// TwinCAT 3 PLC project Untitled1
// ProgramVersion: 3.1.4026.19
// libraries:
//   Tc2_Standard, * (Beckhoff Automation GmbH)
//   Tc2_System, * (Beckhoff Automation GmbH)
// project tree:
//   DUTs/ ST_Chiller_Reads.TcDUT, ST_Alarms.TcDUT (not stored), ST_Control.TcDUT, ST_Chiller_Writes.TcDUT, ST_States.TcDUT (not stored), ST_Value0.TcDUT, ST_Value1.TcDUT (not stored)
//   GVLs/ GVL_Lauda.TcGVL
//   / PlcTask.TcTTO
//   POUs/ FB_Chiller.TcPOU, MAIN.TcPOU (not stored)
// real-time tasks:
//   TASK PlcTask: cycle T#10ms, priority 20, ADS port 350
//   TASK Task_Profinet: cycle T#1ms, priority 1, ADS port 301
// I/O:
//   DEVICE Device 1 (Profinet Controller CCAT (RT)), AmsNetId 5.155.185.217.2.1
//     abx-prt [HMS Industrial Networks This Device Access Point supports RT communication Anybus X-gateway]
//       modules: Term 1 (DAP Module), Term 2 (Output 002 bytes), Term 3 (Output 032 bytes), Term 4 (Input 004 bytes), Term 5 (Input 064 bytes), Term 6 (Input 032 bytes), Term 7 (Input 016 bytes)
// variable links:
//   Untitled1/Untitled1 Instance <-> Device 1 (Profinet Controller CCAT (RT))/abx-prt
//     PlcTask Inputs/GVL_Lauda.LaudaChillerReads.ChilleStatesIn.V50011On <-> API/Term 4 (Input 004 bytes)/Subterm 6 (Input 004 bytes)/Inputs/Input[0] @bit 2
//     PlcTask Inputs/GVL_Lauda.LaudaChillerReads.ChilleStatesIn.commonFault <-> API/Term 4 (Input 004 bytes)/Subterm 6 (Input 004 bytes)/Inputs/Input[1] @bit 1
//     PlcTask Inputs/GVL_Lauda.LaudaChillerReads.ChilleStatesIn.commonWarning <-> API/Term 4 (Input 004 bytes)/Subterm 6 (Input 004 bytes)/Inputs/Input[1] @bit 2
//     PlcTask Inputs/GVL_Lauda.LaudaChillerReads.ChilleStatesIn.cooling <-> API/Term 4 (Input 004 bytes)/Subterm 6 (Input 004 bytes)/Inputs/Input[0] @bit 7
//     PlcTask Inputs/GVL_Lauda.LaudaChillerReads.ChilleStatesIn.criticalError <-> API/Term 4 (Input 004 bytes)/Subterm 6 (Input 004 bytes)/Inputs/Input[1] @bit 3
//     PlcTask Inputs/GVL_Lauda.LaudaChillerReads.ChilleStatesIn.filling <-> API/Term 4 (Input 004 bytes)/Subterm 6 (Input 004 bytes)/Inputs/Input[0] @bit 5
//     PlcTask Inputs/GVL_Lauda.LaudaChillerReads.ChilleStatesIn.heating <-> API/Term 4 (Input 004 bytes)/Subterm 6 (Input 004 bytes)/Inputs/Input[0] @bit 6
//     PlcTask Inputs/GVL_Lauda.LaudaChillerReads.ChilleStatesIn.operation <-> API/Term 4 (Input 004 bytes)/Subterm 6 (Input 004 bytes)/Inputs/Input[0] @bit 1
//     PlcTask Inputs/GVL_Lauda.LaudaChillerReads.ChilleStatesIn.ready <-> API/Term 4 (Input 004 bytes)/Subterm 6 (Input 004 bytes)/Inputs/Input[1]
//     PlcTask Inputs/GVL_Lauda.LaudaChillerReads.ChilleStatesIn.remote <-> API/Term 4 (Input 004 bytes)/Subterm 6 (Input 004 bytes)/Inputs/Input[0] @bit 4
//     PlcTask Inputs/GVL_Lauda.LaudaChillerReads.ChilleStatesIn.v60011On <-> API/Term 4 (Input 004 bytes)/Subterm 6 (Input 004 bytes)/Inputs/Input[0] @bit 3
//     PlcTask Inputs/GVL_Lauda.LaudaChillerReads.ChilleStatesIn.watchdog <-> API/Term 4 (Input 004 bytes)/Subterm 6 (Input 004 bytes)/Inputs/Input[0]
//     PlcTask Inputs/GVL_Lauda.LaudaChillerReads.ChillerAlarmsIn._230VAC <-> API/Term 7 (Input 016 bytes)/Subterm 9 (Input 016 bytes)/Inputs/Input[0] @bit 2
//     PlcTask Inputs/GVL_Lauda.LaudaChillerReads.ChillerAlarmsIn._24VDC <-> API/Term 7 (Input 016 bytes)/Subterm 9 (Input 016 bytes)/Inputs/Input[0] @bit 3
//     PlcTask Inputs/GVL_Lauda.LaudaChillerReads.ChillerAlarmsIn._24VDC_Puffer <-> API/Term 7 (Input 016 bytes)/Subterm 9 (Input 016 bytes)/Inputs/Input[0] @bit 4
//     PlcTask Inputs/GVL_Lauda.LaudaChillerReads.ChillerAlarmsIn.communicationDCS <-> API/Term 7 (Input 016 bytes)/Subterm 9 (Input 016 bytes)/Inputs/Input[0] @bit 6
//     PlcTask Inputs/GVL_Lauda.LaudaChillerReads.ChillerAlarmsIn.eStopExternal <-> API/Term 7 (Input 016 bytes)/Subterm 9 (Input 016 bytes)/Inputs/Input[0] @bit 1
//     PlcTask Inputs/GVL_Lauda.LaudaChillerReads.ChillerAlarmsIn.eStopInternal <-> API/Term 7 (Input 016 bytes)/Subterm 9 (Input 016 bytes)/Inputs/Input[0]
//     PlcTask Inputs/GVL_Lauda.LaudaChillerReads.ChillerAlarmsIn.profinet <-> API/Term 7 (Input 016 bytes)/Subterm 9 (Input 016 bytes)/Inputs/Input[0] @bit 5
//     PlcTask Inputs/GVL_Lauda.LaudaChillerReads.ChillerAlarmsIn.sfSafteySPS <-> API/Term 7 (Input 016 bytes)/Subterm 9 (Input 016 bytes)/Inputs/Input[0] @bit 7
//     PlcTask Inputs/GVL_Lauda.LaudaChillerReads.ChillerValuesIn.B10011 @bit 24 <-> API/Term 5 (Input 064 bytes)/Subterm 7 (Input 064 bytes)/Inputs/Input[4]
//     PlcTask Inputs/GVL_Lauda.LaudaChillerReads.ChillerValuesIn.B10011 @bit 16 <-> API/Term 5 (Input 064 bytes)/Subterm 7 (Input 064 bytes)/Inputs/Input[5]
//     PlcTask Inputs/GVL_Lauda.LaudaChillerReads.ChillerValuesIn.B10011 @bit 8 <-> API/Term 5 (Input 064 bytes)/Subterm 7 (Input 064 bytes)/Inputs/Input[6]
//     PlcTask Inputs/GVL_Lauda.LaudaChillerReads.ChillerValuesIn.B10511 @bit 8 <-> API/Term 5 (Input 064 bytes)/Subterm 7 (Input 064 bytes)/Inputs/Input[10]
//     PlcTask Inputs/GVL_Lauda.LaudaChillerReads.ChillerValuesIn.B10511 @bit 24 <-> API/Term 5 (Input 064 bytes)/Subterm 7 (Input 064 bytes)/Inputs/Input[8]
//     PlcTask Inputs/GVL_Lauda.LaudaChillerReads.ChillerValuesIn.B10511 @bit 16 <-> API/Term 5 (Input 064 bytes)/Subterm 7 (Input 064 bytes)/Inputs/Input[9]
//     PlcTask Inputs/GVL_Lauda.LaudaChillerReads.ChillerValuesIn.B10512 @bit 24 <-> API/Term 5 (Input 064 bytes)/Subterm 7 (Input 064 bytes)/Inputs/Input[12]
//     PlcTask Inputs/GVL_Lauda.LaudaChillerReads.ChillerValuesIn.B10512 @bit 16 <-> API/Term 5 (Input 064 bytes)/Subterm 7 (Input 064 bytes)/Inputs/Input[13]
//     PlcTask Inputs/GVL_Lauda.LaudaChillerReads.ChillerValuesIn.B10512 @bit 8 <-> API/Term 5 (Input 064 bytes)/Subterm 7 (Input 064 bytes)/Inputs/Input[14]
//     PlcTask Inputs/GVL_Lauda.LaudaChillerReads.ChillerValuesIn.B14011 @bit 24 <-> API/Term 5 (Input 064 bytes)/Subterm 7 (Input 064 bytes)/Inputs/Input[16]
//     PlcTask Inputs/GVL_Lauda.LaudaChillerReads.ChillerValuesIn.B14011 @bit 16 <-> API/Term 5 (Input 064 bytes)/Subterm 7 (Input 064 bytes)/Inputs/Input[17]
//     PlcTask Inputs/GVL_Lauda.LaudaChillerReads.ChillerValuesIn.B14011 @bit 8 <-> API/Term 5 (Input 064 bytes)/Subterm 7 (Input 064 bytes)/Inputs/Input[18]
//     PlcTask Inputs/GVL_Lauda.LaudaChillerReads.ChillerValuesIn.B16411 @bit 24 <-> API/Term 5 (Input 064 bytes)/Subterm 7 (Input 064 bytes)/Inputs/Input[20]
//     PlcTask Inputs/GVL_Lauda.LaudaChillerReads.ChillerValuesIn.B16411 @bit 16 <-> API/Term 5 (Input 064 bytes)/Subterm 7 (Input 064 bytes)/Inputs/Input[21]
//     PlcTask Inputs/GVL_Lauda.LaudaChillerReads.ChillerValuesIn.B16411 @bit 8 <-> API/Term 5 (Input 064 bytes)/Subterm 7 (Input 064 bytes)/Inputs/Input[22]
//     PlcTask Inputs/GVL_Lauda.LaudaChillerReads.ChillerValuesIn.B18011 @bit 24 <-> API/Term 5 (Input 064 bytes)/Subterm 7 (Input 064 bytes)/Inputs/Input[24]
//     PlcTask Inputs/GVL_Lauda.LaudaChillerReads.ChillerValuesIn.B18011 @bit 16 <-> API/Term 5 (Input 064 bytes)/Subterm 7 (Input 064 bytes)/Inputs/Input[25]
//     PlcTask Inputs/GVL_Lauda.LaudaChillerReads.ChillerValuesIn.B18011 @bit 8 <-> API/Term 5 (Input 064 bytes)/Subterm 7 (Input 064 bytes)/Inputs/Input[26]
//     PlcTask Inputs/GVL_Lauda.LaudaChillerReads.ChillerValuesIn.B55111 @bit 24 <-> API/Term 5 (Input 064 bytes)/Subterm 7 (Input 064 bytes)/Inputs/Input[28]
//     PlcTask Inputs/GVL_Lauda.LaudaChillerReads.ChillerValuesIn.B55111 @bit 16 <-> API/Term 5 (Input 064 bytes)/Subterm 7 (Input 064 bytes)/Inputs/Input[29]
//     PlcTask Inputs/GVL_Lauda.LaudaChillerReads.ChillerValuesIn.B55111 @bit 8 <-> API/Term 5 (Input 064 bytes)/Subterm 7 (Input 064 bytes)/Inputs/Input[30]
//     PlcTask Inputs/GVL_Lauda.LaudaChillerReads.ChillerValuesIn.B55211 @bit 24 <-> API/Term 5 (Input 064 bytes)/Subterm 7 (Input 064 bytes)/Inputs/Input[32]
//     PlcTask Inputs/GVL_Lauda.LaudaChillerReads.ChillerValuesIn.B55211 @bit 16 <-> API/Term 5 (Input 064 bytes)/Subterm 7 (Input 064 bytes)/Inputs/Input[33]
//     PlcTask Inputs/GVL_Lauda.LaudaChillerReads.ChillerValuesIn.B55211 @bit 8 <-> API/Term 5 (Input 064 bytes)/Subterm 7 (Input 064 bytes)/Inputs/Input[34]
//     PlcTask Inputs/GVL_Lauda.LaudaChillerReads.ChillerValuesIn.B55811 @bit 24 <-> API/Term 5 (Input 064 bytes)/Subterm 7 (Input 064 bytes)/Inputs/Input[36]
//     PlcTask Inputs/GVL_Lauda.LaudaChillerReads.ChillerValuesIn.B55811 @bit 16 <-> API/Term 5 (Input 064 bytes)/Subterm 7 (Input 064 bytes)/Inputs/Input[37]
//     PlcTask Inputs/GVL_Lauda.LaudaChillerReads.ChillerValuesIn.B55811 @bit 8 <-> API/Term 5 (Input 064 bytes)/Subterm 7 (Input 064 bytes)/Inputs/Input[38]
//     PlcTask Inputs/GVL_Lauda.LaudaChillerReads.ChillerValuesIn.B56511 @bit 24 <-> API/Term 5 (Input 064 bytes)/Subterm 7 (Input 064 bytes)/Inputs/Input[40]
//     PlcTask Inputs/GVL_Lauda.LaudaChillerReads.ChillerValuesIn.B56511 @bit 16 <-> API/Term 5 (Input 064 bytes)/Subterm 7 (Input 064 bytes)/Inputs/Input[41]
//     PlcTask Inputs/GVL_Lauda.LaudaChillerReads.ChillerValuesIn.B56511 @bit 8 <-> API/Term 5 (Input 064 bytes)/Subterm 7 (Input 064 bytes)/Inputs/Input[42]
//     PlcTask Inputs/GVL_Lauda.LaudaChillerReads.ChillerValuesIn.B56811 @bit 24 <-> API/Term 5 (Input 064 bytes)/Subterm 7 (Input 064 bytes)/Inputs/Input[44]
//     PlcTask Inputs/GVL_Lauda.LaudaChillerReads.ChillerValuesIn.B56811 @bit 16 <-> API/Term 5 (Input 064 bytes)/Subterm 7 (Input 064 bytes)/Inputs/Input[45]
//     PlcTask Inputs/GVL_Lauda.LaudaChillerReads.ChillerValuesIn.B56811 @bit 8 <-> API/Term 5 (Input 064 bytes)/Subterm 7 (Input 064 bytes)/Inputs/Input[46]
//     PlcTask Inputs/GVL_Lauda.LaudaChillerReads.ChillerValuesIn.B57311 @bit 24 <-> API/Term 5 (Input 064 bytes)/Subterm 7 (Input 064 bytes)/Inputs/Input[48]
//     PlcTask Inputs/GVL_Lauda.LaudaChillerReads.ChillerValuesIn.B57311 @bit 16 <-> API/Term 5 (Input 064 bytes)/Subterm 7 (Input 064 bytes)/Inputs/Input[49]
//     PlcTask Inputs/GVL_Lauda.LaudaChillerReads.ChillerValuesIn.B57311 @bit 8 <-> API/Term 5 (Input 064 bytes)/Subterm 7 (Input 064 bytes)/Inputs/Input[50]
//     PlcTask Inputs/GVL_Lauda.LaudaChillerReads.ChillerValuesIn.B65111 @bit 24 <-> API/Term 5 (Input 064 bytes)/Subterm 7 (Input 064 bytes)/Inputs/Input[52]
//     PlcTask Inputs/GVL_Lauda.LaudaChillerReads.ChillerValuesIn.B65111 @bit 16 <-> API/Term 5 (Input 064 bytes)/Subterm 7 (Input 064 bytes)/Inputs/Input[53]
//     PlcTask Inputs/GVL_Lauda.LaudaChillerReads.ChillerValuesIn.B65111 @bit 8 <-> API/Term 5 (Input 064 bytes)/Subterm 7 (Input 064 bytes)/Inputs/Input[54]
//     PlcTask Inputs/GVL_Lauda.LaudaChillerReads.ChillerValuesIn.B65211 @bit 24 <-> API/Term 5 (Input 064 bytes)/Subterm 7 (Input 064 bytes)/Inputs/Input[56]
//     PlcTask Inputs/GVL_Lauda.LaudaChillerReads.ChillerValuesIn.B65211 @bit 16 <-> API/Term 5 (Input 064 bytes)/Subterm 7 (Input 064 bytes)/Inputs/Input[57]
//     PlcTask Inputs/GVL_Lauda.LaudaChillerReads.ChillerValuesIn.B65211 @bit 8 <-> API/Term 5 (Input 064 bytes)/Subterm 7 (Input 064 bytes)/Inputs/Input[58]
//     PlcTask Inputs/GVL_Lauda.LaudaChillerReads.ChillerValuesIn.B65511 @bit 24 <-> API/Term 5 (Input 064 bytes)/Subterm 7 (Input 064 bytes)/Inputs/Input[60]
//     PlcTask Inputs/GVL_Lauda.LaudaChillerReads.ChillerValuesIn.B65511 @bit 16 <-> API/Term 5 (Input 064 bytes)/Subterm 7 (Input 064 bytes)/Inputs/Input[61]
//     PlcTask Inputs/GVL_Lauda.LaudaChillerReads.ChillerValuesIn.B65511 @bit 8 <-> API/Term 5 (Input 064 bytes)/Subterm 7 (Input 064 bytes)/Inputs/Input[62]
//     PlcTask Inputs/GVL_Lauda.LaudaChillerReads.ChillerValuesIn.B65811 @bit 24 <-> API/Term 6 (Input 032 bytes)/Subterm 8 (Input 032 bytes)/Inputs/Input[0]
//     PlcTask Inputs/GVL_Lauda.LaudaChillerReads.ChillerValuesIn.B65811 @bit 16 <-> API/Term 6 (Input 032 bytes)/Subterm 8 (Input 032 bytes)/Inputs/Input[1]
//     PlcTask Inputs/GVL_Lauda.LaudaChillerReads.ChillerValuesIn.B65811 @bit 8 <-> API/Term 6 (Input 032 bytes)/Subterm 8 (Input 032 bytes)/Inputs/Input[2]
//     PlcTask Inputs/GVL_Lauda.LaudaChillerReads.ChillerValuesIn.B66511 @bit 24 <-> API/Term 6 (Input 032 bytes)/Subterm 8 (Input 032 bytes)/Inputs/Input[4]
//     PlcTask Inputs/GVL_Lauda.LaudaChillerReads.ChillerValuesIn.B66511 @bit 16 <-> API/Term 6 (Input 032 bytes)/Subterm 8 (Input 032 bytes)/Inputs/Input[5]
//     PlcTask Inputs/GVL_Lauda.LaudaChillerReads.ChillerValuesIn.B66511 @bit 8 <-> API/Term 6 (Input 032 bytes)/Subterm 8 (Input 032 bytes)/Inputs/Input[6]
//     PlcTask Inputs/GVL_Lauda.LaudaChillerReads.ChillerValuesIn.B66811 @bit 8 <-> API/Term 6 (Input 032 bytes)/Subterm 8 (Input 032 bytes)/Inputs/Input[10]
//     PlcTask Inputs/GVL_Lauda.LaudaChillerReads.ChillerValuesIn.B66811 @bit 24 <-> API/Term 6 (Input 032 bytes)/Subterm 8 (Input 032 bytes)/Inputs/Input[8]
//     PlcTask Inputs/GVL_Lauda.LaudaChillerReads.ChillerValuesIn.B66811 @bit 16 <-> API/Term 6 (Input 032 bytes)/Subterm 8 (Input 032 bytes)/Inputs/Input[9]
//     PlcTask Inputs/GVL_Lauda.LaudaChillerReads.ChillerValuesIn.B67311 @bit 24 <-> API/Term 6 (Input 032 bytes)/Subterm 8 (Input 032 bytes)/Inputs/Input[12]
//     PlcTask Inputs/GVL_Lauda.LaudaChillerReads.ChillerValuesIn.B67311 @bit 16 <-> API/Term 6 (Input 032 bytes)/Subterm 8 (Input 032 bytes)/Inputs/Input[13]
//     PlcTask Inputs/GVL_Lauda.LaudaChillerReads.ChillerValuesIn.B67311 @bit 8 <-> API/Term 6 (Input 032 bytes)/Subterm 8 (Input 032 bytes)/Inputs/Input[14]
//     PlcTask Inputs/GVL_Lauda.LaudaChillerReads.ChillerValuesIn.B10011 <-> API/Term 5 (Input 064 bytes)/Subterm 7 (Input 064 bytes)/Inputs/Input[7]
//     PlcTask Inputs/GVL_Lauda.LaudaChillerReads.ChillerValuesIn.B10511 <-> API/Term 5 (Input 064 bytes)/Subterm 7 (Input 064 bytes)/Inputs/Input[11]
//     PlcTask Inputs/GVL_Lauda.LaudaChillerReads.ChillerValuesIn.B10512 <-> API/Term 5 (Input 064 bytes)/Subterm 7 (Input 064 bytes)/Inputs/Input[15]
//     PlcTask Inputs/GVL_Lauda.LaudaChillerReads.ChillerValuesIn.B14011 <-> API/Term 5 (Input 064 bytes)/Subterm 7 (Input 064 bytes)/Inputs/Input[19]
//     PlcTask Inputs/GVL_Lauda.LaudaChillerReads.ChillerValuesIn.B16411 <-> API/Term 5 (Input 064 bytes)/Subterm 7 (Input 064 bytes)/Inputs/Input[23]
//     PlcTask Inputs/GVL_Lauda.LaudaChillerReads.ChillerValuesIn.B18011 <-> API/Term 5 (Input 064 bytes)/Subterm 7 (Input 064 bytes)/Inputs/Input[27]
//     PlcTask Inputs/GVL_Lauda.LaudaChillerReads.ChillerValuesIn.B55111 <-> API/Term 5 (Input 064 bytes)/Subterm 7 (Input 064 bytes)/Inputs/Input[31]
//     PlcTask Inputs/GVL_Lauda.LaudaChillerReads.ChillerValuesIn.B55211 <-> API/Term 5 (Input 064 bytes)/Subterm 7 (Input 064 bytes)/Inputs/Input[35]
//     PlcTask Inputs/GVL_Lauda.LaudaChillerReads.ChillerValuesIn.B55811 <-> API/Term 5 (Input 064 bytes)/Subterm 7 (Input 064 bytes)/Inputs/Input[39]
//     PlcTask Inputs/GVL_Lauda.LaudaChillerReads.ChillerValuesIn.B56511 <-> API/Term 5 (Input 064 bytes)/Subterm 7 (Input 064 bytes)/Inputs/Input[43]
//     PlcTask Inputs/GVL_Lauda.LaudaChillerReads.ChillerValuesIn.B56811 <-> API/Term 5 (Input 064 bytes)/Subterm 7 (Input 064 bytes)/Inputs/Input[47]
//     PlcTask Inputs/GVL_Lauda.LaudaChillerReads.ChillerValuesIn.B57311 <-> API/Term 5 (Input 064 bytes)/Subterm 7 (Input 064 bytes)/Inputs/Input[51]
//     PlcTask Inputs/GVL_Lauda.LaudaChillerReads.ChillerValuesIn.B65111 <-> API/Term 5 (Input 064 bytes)/Subterm 7 (Input 064 bytes)/Inputs/Input[55]
//     PlcTask Inputs/GVL_Lauda.LaudaChillerReads.ChillerValuesIn.B65211 <-> API/Term 5 (Input 064 bytes)/Subterm 7 (Input 064 bytes)/Inputs/Input[59]
//     PlcTask Inputs/GVL_Lauda.LaudaChillerReads.ChillerValuesIn.B65511 <-> API/Term 5 (Input 064 bytes)/Subterm 7 (Input 064 bytes)/Inputs/Input[63]
//     PlcTask Inputs/GVL_Lauda.LaudaChillerReads.ChillerValuesIn.B65811 <-> API/Term 6 (Input 032 bytes)/Subterm 8 (Input 032 bytes)/Inputs/Input[3]
//     PlcTask Inputs/GVL_Lauda.LaudaChillerReads.ChillerValuesIn.B66511 <-> API/Term 6 (Input 032 bytes)/Subterm 8 (Input 032 bytes)/Inputs/Input[7]
//     PlcTask Inputs/GVL_Lauda.LaudaChillerReads.ChillerValuesIn.B66811 <-> API/Term 6 (Input 032 bytes)/Subterm 8 (Input 032 bytes)/Inputs/Input[11]
//     PlcTask Inputs/GVL_Lauda.LaudaChillerReads.ChillerValuesIn.B67311 <-> API/Term 6 (Input 032 bytes)/Subterm 8 (Input 032 bytes)/Inputs/Input[15]
//     PlcTask Inputs/GVL_Lauda.LaudaChillerReads.ChillerValuesIn.N10011 @bit 24 <-> API/Term 6 (Input 032 bytes)/Subterm 8 (Input 032 bytes)/Inputs/Input[16]
//     PlcTask Inputs/GVL_Lauda.LaudaChillerReads.ChillerValuesIn.N10011 @bit 16 <-> API/Term 6 (Input 032 bytes)/Subterm 8 (Input 032 bytes)/Inputs/Input[17]
//     PlcTask Inputs/GVL_Lauda.LaudaChillerReads.ChillerValuesIn.N10011 @bit 8 <-> API/Term 6 (Input 032 bytes)/Subterm 8 (Input 032 bytes)/Inputs/Input[18]
//     PlcTask Inputs/GVL_Lauda.LaudaChillerReads.ChillerValuesIn.N10011 <-> API/Term 6 (Input 032 bytes)/Subterm 8 (Input 032 bytes)/Inputs/Input[19]
//     PlcTask Inputs/GVL_Lauda.LaudaChillerReads.ChillerValuesIn.actualSetpoint @bit 24 <-> API/Term 5 (Input 064 bytes)/Subterm 7 (Input 064 bytes)/Inputs/Input[0]
//     PlcTask Inputs/GVL_Lauda.LaudaChillerReads.ChillerValuesIn.actualSetpoint @bit 16 <-> API/Term 5 (Input 064 bytes)/Subterm 7 (Input 064 bytes)/Inputs/Input[1]
//     PlcTask Inputs/GVL_Lauda.LaudaChillerReads.ChillerValuesIn.actualSetpoint @bit 8 <-> API/Term 5 (Input 064 bytes)/Subterm 7 (Input 064 bytes)/Inputs/Input[2]
//     PlcTask Inputs/GVL_Lauda.LaudaChillerReads.ChillerValuesIn.actualSetpoint <-> API/Term 5 (Input 064 bytes)/Subterm 7 (Input 064 bytes)/Inputs/Input[3]
//     PlcTask Outputs/GVL_Lauda.LaudaChillerWrites.controlOut.remote <-> API/Term 2 (Output 002 bytes)/Subterm 4 (Output 002 bytes)/Outputs/Output[0] @bit 3
//     PlcTask Outputs/GVL_Lauda.LaudaChillerWrites.controlOut.reset <-> API/Term 2 (Output 002 bytes)/Subterm 4 (Output 002 bytes)/Outputs/Output[0] @bit 2
//     PlcTask Outputs/GVL_Lauda.LaudaChillerWrites.controlOut.start_Stop <-> API/Term 2 (Output 002 bytes)/Subterm 4 (Output 002 bytes)/Outputs/Output[0] @bit 1
//     PlcTask Outputs/GVL_Lauda.LaudaChillerWrites.controlOut.watchdog <-> API/Term 2 (Output 002 bytes)/Subterm 4 (Output 002 bytes)/Outputs/Output[0]
//     PlcTask Outputs/GVL_Lauda.LaudaChillerWrites.valueOut.speedPumpN14011 <-> API/Term 3 (Output 032 bytes)/Subterm 5 (Output 032 bytes)/Outputs/Output[16]
//     PlcTask Outputs/GVL_Lauda.LaudaChillerWrites.valueOut.speedPumpN14011 @bit 8 <-> API/Term 3 (Output 032 bytes)/Subterm 5 (Output 032 bytes)/Outputs/Output[17]
//     PlcTask Outputs/GVL_Lauda.LaudaChillerWrites.valueOut.speedPumpN14011 @bit 16 <-> API/Term 3 (Output 032 bytes)/Subterm 5 (Output 032 bytes)/Outputs/Output[18]
//     PlcTask Outputs/GVL_Lauda.LaudaChillerWrites.valueOut.speedPumpN14011 @bit 24 <-> API/Term 3 (Output 032 bytes)/Subterm 5 (Output 032 bytes)/Outputs/Output[19]
//     PlcTask Outputs/GVL_Lauda.LaudaChillerWrites.valueOut.tempSetpointN10011 <-> API/Term 3 (Output 032 bytes)/Subterm 5 (Output 032 bytes)/Outputs/Output[0]
//     PlcTask Outputs/GVL_Lauda.LaudaChillerWrites.valueOut.tempSetpointN10011 @bit 8 <-> API/Term 3 (Output 032 bytes)/Subterm 5 (Output 032 bytes)/Outputs/Output[1]
//     PlcTask Outputs/GVL_Lauda.LaudaChillerWrites.valueOut.tempSetpointN10011 @bit 16 <-> API/Term 3 (Output 032 bytes)/Subterm 5 (Output 032 bytes)/Outputs/Output[2]
//     PlcTask Outputs/GVL_Lauda.LaudaChillerWrites.valueOut.tempSetpointN10011 @bit 24 <-> API/Term 3 (Output 032 bytes)/Subterm 5 (Output 032 bytes)/Outputs/Output[3]

CONFIGURATION Untitled1
    RESOURCE PLC ON TwinCAT3
        TASK PlcTask(INTERVAL := T#10ms, PRIORITY := 20);
        PROGRAM MAIN WITH PlcTask : MAIN;
    END_RESOURCE
END_CONFIGURATION

// ---- DUTs/ST_Chiller_Reads.TcDUT
{attribute 'pack_mode' := '1'}
TYPE ST_Chiller_Reads :
STRUCT
	ChilleStatesIn  : ST_States;
	ChillerValuesIn : ST_Value1;
	ChillerAlarmsIn : ST_Alarms;
END_STRUCT
END_TYPE

// ---- DUTs/ST_Control.TcDUT
{attribute 'pack_mode' := '1'}
TYPE ST_Control :
STRUCT
	watchdog AT %Q*: BOOL;
	start_Stop AT %Q* : BOOL;
	reset AT %Q* : BOOL;
	remote AT %Q* : BOOL;
END_STRUCT
END_TYPE

// ---- DUTs/ST_Chiller_Writes.TcDUT
{attribute 'pack_mode' := '1'}
TYPE ST_Chiller_Writes :
STRUCT
	controlOut : ST_Control;
	valueOut : ST_Value0;
END_STRUCT
END_TYPE

// ---- DUTs/ST_Value0.TcDUT
{attribute 'pack_mode' := '1'}
TYPE ST_Value0 :
STRUCT
	tempSetpointN10011 AT %Q* : REAL;
	speedPumpN14011  AT %Q*: REAL;
END_STRUCT
END_TYPE

// ---- GVLs/GVL_Lauda.TcGVL
{attribute 'qualified_only'}
VAR_GLOBAL
	LaudaChillerWrites : ST_Chiller_Writes;
	LaudaChillerReads : ST_Chiller_Reads;
END_VAR

// ---- POUs/FB_Chiller.TcPOU
FUNCTION_BLOCK FB_Chiller
VAR_INPUT
END_VAR
VAR_OUTPUT
END_VAR
VAR
END_VAR

END_FUNCTION_BLOCK
